# B&R Automation Studio project 305841_E00002_AM_0 (part 4)

#### Init.st
```iecst
PROGRAM _INIT

  // TODO: Security levels. For now just set as operator so OM SM can be programmed
  operatingMode.SecurityLevel := SL_OPERATOR;

  // EMO Reset time
  timeEStopResetAllow := T#10s;
  timeResetPulse := T#1s;

  // Init to create variables
  // If values are only mapped, and not used in logic anywhere, the compiler does not
  // create them. They are not available to
  // the HMI, and the compiler also complains about
  // them being declared but not used
  fs_AllSMsOk := FALSE;
  fs_EmoCmd := FALSE;
  fs_EmoOwsActive := FALSE;
  fs_EmoOwsOk := FALSE;
  // pendant signals are mapped into pendant structure
  // fs_EmoPendantActive := FALSE;
  // fs_EmoPendantOk := FALSE;
  // fs_AllowPendantMoves := FALSE;
  fs_KeyswitchInRun := FALSE;
  fs_KeyswitchOk := FALSE;
  fs_InSafeMode := FALSE;
  fs_StartPbActive := FALSE;
  fs_StartPbOk := FALSE;
  fs_StopPbActive := FALSE;
  fs_StopPbOk := FALSE;
  fs_CfGateClosedLocked := FALSE;
  fs_CfGateClosedOk := FALSE;

  ts_ResetEStop := FALSE;
  ts_ResetSafeMC := FALSE;

  // Init process req fb
  procHmiProcessReqs._I_ProcessReqs := ADR(hmiProcessReqs);
  procHmiProcessReqs._I_WpCfg := ADR(gr_CfgCurrent);
  // use the base (element 0) address for these arrays. Element
  // positions will be calculated and accessed within the function
  procHmiProcessReqs._I_pLibraryAxesReqs := ADR(hmiLibraryAxisReqs);
  procHmiProcessReqs._I_pAxis := ADR(axes);
  procHmiProcessReqs._I_pAxisPositionLimits := ADR(gr_AxisPositionLimits);

  // Init manual mode requests
  hmiLibraryAxisReqs[AD_SPINDLE].axisNo := DINT_TO_USINT(AD_SPINDLE);
  hmiMachineAxisReqs[AD_SPINDLE].axisNo := DINT_TO_USINT(AD_SPINDLE);
  hmiMachineAxisReqs[AD_SPINDLE].axisDesignation := AD_SPINDLE;
  procManualAxisReqsSpindle._I_Axis := ADR(axes[AD_SPINDLE]);
  procManualAxisReqsSpindle._I_SlaveAxis := ADR(axes[axes[AD_SPINDLE].CouplingParameters.SlaveAxisNo]);
  procManualAxisReqsSpindle._I_LibraryAxisReqs := ADR(hmiLibraryAxisReqs[AD_SPINDLE]);
  procManualAxisReqsSpindle._I_MachineAxisReqs := ADR(hmiMachineAxisReqs[AD_SPINDLE]);
  procManualAxisReqsSpindle._I_AxisPositionLimits := ADR(gr_AxisPositionLimits[AD_SPINDLE]);

  // Outer Eccentric
  hmiLibraryAxisReqs[AD_OUTER_ECCENTRIC].axisNo := DINT_TO_USINT(AD_OUTER_ECCENTRIC);
  hmiMachineAxisReqs[AD_OUTER_ECCENTRIC].axisNo := DINT_TO_USINT(AD_OUTER_ECCENTRIC);
  hmiMachineAxisReqs[AD_OUTER_ECCENTRIC].axisDesignation := AD_OUTER_ECCENTRIC;
  procManualAxisReqsOutE._I_Axis := ADR(axes[AD_OUTER_ECCENTRIC]);
  procManualAxisReqsOutE._I_SlaveAxis := ADR(axes[axes[AD_OUTER_ECCENTRIC].CouplingParameters.SlaveAxisNo]);
  procManualAxisReqsOutE._I_LibraryAxisReqs := ADR(hmiLibraryAxisReqs[AD_OUTER_ECCENTRIC]);
  procManualAxisReqsOutE._I_MachineAxisReqs:= ADR(hmiMachineAxisReqs[AD_OUTER_ECCENTRIC]);
  procManualAxisReqsOutE._I_AxisPositionLimits := ADR(gr_AxisPositionLimits[AD_OUTER_ECCENTRIC]);

  // Inner Eccentric
  hmiLibraryAxisReqs[AD_INNER_ECCENTRIC].axisNo := DINT_TO_USINT(AD_INNER_ECCENTRIC);
  hmiMachineAxisReqs[AD_INNER_ECCENTRIC].axisNo := DINT_TO_USINT(AD_INNER_ECCENTRIC);
  hmiMachineAxisReqs[AD_INNER_ECCENTRIC].axisDesignation := AD_INNER_ECCENTRIC;
  procManualAxisReqsInE._I_Axis := ADR(axes[AD_INNER_ECCENTRIC]);
  procManualAxisReqsInE._I_SlaveAxis := ADR(axes[axes[AD_INNER_ECCENTRIC].CouplingParameters.SlaveAxisNo]);
  procManualAxisReqsInE._I_LibraryAxisReqs := ADR(hmiLibraryAxisReqs[AD_INNER_ECCENTRIC]);
  procManualAxisReqsInE._I_MachineAxisReqs := ADR(hmiMachineAxisReqs[AD_INNER_ECCENTRIC]);
  procManualAxisReqsInE._I_AxisPositionLimits := ADR(gr_AxisPositionLimits[AD_INNER_ECCENTRIC]);

  // Z
  hmiLibraryAxisReqs[AD_Z].axisNo := DINT_TO_USINT(AD_Z);
  hmiMachineAxisReqs[AD_Z].axisNo := DINT_TO_USINT(AD_Z);
  hmiMachineAxisReqs[AD_Z].axisDesignation := AD_Z;
  procManualAxisReqsZ._I_Axis := ADR(axes[AD_Z]);
  procManualAxisReqsZ._I_SlaveAxis := ADR(axes[axes[AD_Z].CouplingParameters.SlaveAxisNo]);
  procManualAxisReqsZ._I_LibraryAxisReqs := ADR(hmiLibraryAxisReqs[AD_Z]);
  procManualAxisReqsZ._I_MachineAxisReqs := ADR(hmiMachineAxisReqs[AD_Z]);
  procManualAxisReqsZ._I_AxisPositionLimits := ADR(gr_AxisPositionLimits[AD_Z]);

  // Handwheel (Axis 7)
  hmiLibraryAxisReqs[AD_HANDWHEEL].axisNo := DINT_TO_USINT(AD_HANDWHEEL);
  hmiMachineAxisReqs[AD_HANDWHEEL].axisNo := DINT_TO_USINT(AD_HANDWHEEL);
  hmiMachineAxisReqs[AD_HANDWHEEL].axisDesignation := AD_HANDWHEEL;
  procManualAxisReqsHw._I_Axis := ADR(axes[AD_HANDWHEEL]);
  procManualAxisReqsHw._I_SlaveAxis := ADR(axes[axes[AD_HANDWHEEL].CouplingParameters.SlaveAxisNo]);
  procManualAxisReqsHw._I_LibraryAxisReqs := ADR(hmiLibraryAxisReqs[AD_HANDWHEEL]);
  procManualAxisReqsHw._I_MachineAxisReqs := ADR(hmiMachineAxisReqs[AD_HANDWHEEL]);
  procManualAxisReqsHw._I_AxisPositionLimits := ADR(gr_AxisPositionLimits[AD_HANDWHEEL]);

  // Cutting fluid VFD (Axis 8)
  hmiLibraryAxisReqs[AD_CF_VFD].axisNo := DINT_TO_USINT(AD_CF_VFD);
  hmiMachineAxisReqs[AD_CF_VFD].axisNo := DINT_TO_USINT(AD_CF_VFD);
  hmiMachineAxisReqs[AD_CF_VFD].axisDesignation := AD_CF_VFD;
  procManualAxisReqsCfVfd._I_Axis := ADR(axes[AD_CF_VFD]);
  procManualAxisReqsCfVfd._I_SlaveAxis := ADR(axes[axes[AD_CF_VFD].CouplingParameters.SlaveAxisNo]);
  procManualAxisReqsCfVfd._I_LibraryAxisReqs := ADR(hmiLibraryAxisReqs[AD_CF_VFD]);
  procManualAxisReqsCfVfd._I_MachineAxisReqs := ADR(hmiMachineAxisReqs[AD_CF_VFD]);
  procManualAxisReqsCfVfd._I_AxisPositionLimits := ADR(gr_AxisPositionLimits[AD_CF_VFD]);

  // Clear reqs that may result in motion or physical changes to an axis
  ClearMotionReqs;
  // Clear other requests
  ClearNonMotionReqs;

END_PROGRAM
```

#### LocalFunctions.st
```iecst
(* This function block will turn machine specific requests into GaMpMotion library requests,
and the library requests will handled with the motion library.
In this way, there is a cascading mechanism to get machine specific then axis
specific reqeusts processed by standard library functions,
even when process or machine specific things are not known by the library functions.
Note that the HMI binds to value in library axis req (sMot_HmiAxisReqs) for the move
requests, and move params. When controlling an individual axis, these are not machine specific.
This fb handles things like enable/disable choices based on selection, or other machine specific things. *)
FUNCTION_BLOCK fbHandleHmiAxisReq // Condition HMI machine specific requests, and then process them with GaMpMotion library fbProcessHmiAxisReq.
  // Map (decode) HMI move type and then direction that the GAMpMotion library will see.
  // Note the direction and move parameters allowd are be influenced by the move type.
  // Do this before processing the move request so values can be checked or used before issuing a move.

  // Endless Axes, or continuous rotary axes (spindle and eccentrics) in this case,
  // in theory can use pos, neg, or shortest path (NOT supported yet).
  // For absolute moves, but non-continuous axes (Z) don't have a specfied direction for absolute moves -- the
  // direction is inherent to the requested position.
  // Also, an absolute move does not need distance, and a relative move does not need a position.
  // A velocity move does not need either.
  // Set the enable bits of the move direction as appropriate
  IF _I_MachineAxisReqs.moveDesignation = 0 THEN // absolute
    // An absolute move does not use distance, only position
    _I_MachineAxisReqs.moveDistanceEnable := FALSE;
    _I_MachineAxisReqs.movePositionEnable := TRUE;
    // now look at the axis and decied on what directions are allowed.
    IF _I_Axis.isAxisEndless THEN
      // Endless axis, absolute move: forward, backward, and shortest (if supported) are allowed
      _I_MachineAxisReqs.directionPosEnable := TRUE;
      _I_MachineAxisReqs.directionNegEnable := TRUE;
      _I_MachineAxisReqs.directionShortestEnable := FALSE; // could be true, but shortest is not supported yet
      // If the selected direction is shortest, then clear the selection
      IF _I_MachineAxisReqs.direction = 2 THEN
        _I_MachineAxisReqs.direction := -1;
      END_IF;
    ELSE
      // For non-endless axis, direction is inferred by move position, so the operator does not choose it
      // Disable choices and clear the selection
      _I_MachineAxisReqs.directionPosEnable := FALSE;
      _I_MachineAxisReqs.directionNegEnable := FALSE;
      _I_MachineAxisReqs.directionShortestEnable := FALSE;
      _I_MachineAxisReqs.direction := -1;
    END_IF;
  ELSIF _I_MachineAxisReqs.moveDesignation = 1 THEN // relative
    // A relative move does not use position, only distance
    _I_MachineAxisReqs.moveDistanceEnable := TRUE;
    _I_MachineAxisReqs.movePositionEnable := FALSE;
    // All axes, relative move: forward and backward are viable selections
    _I_MachineAxisReqs.directionPosEnable := TRUE;
    _I_MachineAxisReqs.directionNegEnable := TRUE;
    _I_MachineAxisReqs.directionShortestEnable := FALSE;
    // If the selected direction is shortest, then clear the selection
    IF _I_MachineAxisReqs.direction = 2 THEN
      _I_MachineAxisReqs.direction := -1;
    END_IF;
  ELSIF _I_MachineAxisReqs.moveDesignation = 2 THEN // velocity
    // A velocity move does not use position or distance
    _I_MachineAxisReqs.moveDistanceEnable := FALSE;
    _I_MachineAxisReqs.movePositionEnable := FALSE;
    // All axes, velocity move: forward and backward are viable selections
    _I_MachineAxisReqs.directionPosEnable := TRUE;
    _I_MachineAxisReqs.directionNegEnable := TRUE;
    _I_MachineAxisReqs.directionShortestEnable := FALSE;
    // If the selected direction is shortest, then clear the selection
    IF _I_MachineAxisReqs.direction = 2 THEN
      _I_MachineAxisReqs.direction := -1;
    END_IF;
  ELSE
    // Not caught move type (error case).
    // Allow move direction so move type can be determined in the move velocity case
    _I_MachineAxisReqs.moveDistanceEnable := FALSE;
    _I_MachineAxisReqs.movePositionEnable := FALSE;
    _I_MachineAxisReqs.directionPosEnable := FALSE;
    _I_MachineAxisReqs.directionNegEnable := FALSE;
    _I_MachineAxisReqs.directionShortestEnable := FALSE;
    _I_MachineAxisReqs.direction := -1;
  END_IF;

  // Coordinated axis PB enable related

  // Gear In and Cam In
  // There must be a slave axis designated,
  // the axes must be homed and enabled,
  // and these two (gear/cam) are mutually exclusive of each other
  _I_MachineAxisReqs.gearInEnable :=
    _I_Axis.CouplingParameters.SlaveAxisNo <> 0 AND
    _I_Axis.Status.IsHomed AND _I_Axis.Status.IsPoweredOn AND
    _I_SlaveAxis.Status.IsHomed AND _I_SlaveAxis.Status.IsPoweredOn AND
    NOT _I_Axis.fbCamIn.Active;

  _I_MachineAxisReqs.camInEnable :=
    _I_Axis.CouplingParameters.SlaveAxisNo <> 0 AND
    _I_Axis.Status.IsHomed AND _I_Axis.Status.IsPoweredOn AND
    _I_SlaveAxis.Status.IsHomed AND _I_SlaveAxis.Status.IsPoweredOn AND
    NOT _I_Axis.fbGearIn.Active;

  // Disengage enabled if gearing or caming is active
  _I_MachineAxisReqs.disengageEnable := _I_Axis.fbGearIn.Active OR _I_Axis.fbCamIn.Active;

  // Coordinated shift commands cannot be enabled unless:
  // 1) The slave is gear coordinated and InSync
  // 2) The master is moving ?? TODO: verify
  // 3) Phase shift and offset shift are not in progress
  // 4) Cam is not active
  _I_MachineAxisReqs.shiftEnable :=
    _I_Axis.Status.IsGearInSync AND
    //_I_Axis.Status.IsMoveActive AND
    NOT _I_Axis.fbOffsetShift.ShiftStarted AND
    NOT _I_Axis.fbPhaseShift.ShiftStarted AND
    NOT _I_Axis.fbCamIn.Active;

  // Now the direction options should be qualified, set the direction that the GAMpMotion library will see
  _I_LibraryAxisReqs.Direction := fctDecodeHmiDirection(_I_DirectionReq := _I_MachineAxisReqs.direction);

  // Decode the HMI move designation into one the GAMpMotion library will see
  _I_LibraryAxisReqs.moveDesignation := fctDecodeHmiMoveType(
  _I_AxisIsEndless := _I_Axis.isAxisEndless,
  _I_MoveReq := _I_MachineAxisReqs.moveDesignation,
  _I_MoveDirection := _I_LibraryAxisReqs.Direction
  );

  // The move type and direction have now been pre-processed. Call the library function to process the requests.
  procLibraryReq(_I_HmiAxisReq := ADR(_I_LibraryAxisReqs),
                 _I_Axis := ADR(_I_Axis),
                 _I_SlaveAxis := ADR(_I_SlaveAxis),
                 _I_AxisPositionLimits := ADR(_I_AxisPositionLimits),
                 _I_ToleranceZeroDepth := TOL_DEPTH_ZERO_DEG);

END_FUNCTION_BLOCK

(* This function block will turn process requests into GaMpMotion library requests.
The GA Motion Library requests will then be handled by the library.
In this way, there is a cascading mechanism to get process specific
reqeusts processed by standard library functions, even when process specific things
are not known by the library functions.*)
FUNCTION_BLOCK fbHandleHmiProcessReqs (* Turn process specific requests into GaMpMotion library requests. *)
  // Calc structure sizes becuase they will be used several times
  szLibReq := SIZEOF(sMot_HmiAxisReqs);
  szAxis := SIZEOF(sMot_Axis);
  szAxisPosLimits := SIZEOF(sMot_PositionLimits);

  // **** Process Cutting Fluid VFD requests

  // First get the CF structures by address arithmetic
  rLibReqs ACCESS _I_pLibraryAxesReqs + (AD_CF_VFD * szLibReq);
  rAxis ACCESS _I_pAxis + (AD_CF_VFD * szAxis);

  // If the axis is enabled issue moves. Otherwise do nothing.
  // Requests get cleared at the end either way
  IF rAxis.Status.IsPoweredOn THEN
    IF _I_ProcessReqs.cfReqRun THEN
      // TODO: Incorporate pressure control
      // FOR NOW: Use RPM regardless
      IF _I_ProcessReqs.cfIsInPressureControl THEN
        rAxis.MoveParameters.Velocity := _I_ProcessReqs.cfRpmCmd / 60.0; // hmi in rpm, but axis is in rps
      ELSE
        rAxis.MoveParameters.Velocity := _I_ProcessReqs.cfRpmCmd / 60.0; // hmi in rpm, but axis is in rps
      END_IF;
      rAxis.MoveParameters.Direction := mcDIR_POSITIVE;
      rAxis.MoveParameters.Acceleration := _I_WpCfg.cfVfd.accel / 60.0; // hmi in rpm, but axis is in rps
      rAxis.MoveParameters.Deceleration := _I_WpCfg.cfVfd.decel / 60.0; // hmi in rpm, but axis is in rps
      rAxis.Commands.MoveVelocityReq := TRUE;
    END_IF;

    IF _I_ProcessReqs.cfReqStop THEN
      rAxis.MoveParameters.Deceleration := _I_WpCfg.cfVfd.decel;
      rAxis.Commands.HaltReq := TRUE;
    END_IF;

  END_IF;

  // **** Process Z axis requests
  // First get the Z structures by address arithmetic
  rLibReqs ACCESS _I_pLibraryAxesReqs + (AD_Z * szLibReq);
  rAxis ACCESS _I_pAxis + (AD_Z * szAxis);
  // get the slave number, and then calc the memory offset
  slaveNum := rAxis.CouplingParameters.SlaveAxisNo;
  rSlaveAxis ACCESS _I_pAxis + (slaveNum * szAxis);
  rAxisPositionLimits ACCESS _I_pAxisPositionLimits + (AD_Z * szAxisPosLimits);

  // Set position requests. Axis needs to be homed if current position is needed.
  // Requests get cleared at the end either way
  IF _I_ProcessReqs.zReqPosSocUseCurrent AND rAxis.Status.IsHomed THEN // home needed since axis position is used
    _I_WpCfg.zAxis.startOfCutPos := rAxis.Status.Position;
  END_IF;
  IF _I_ProcessReqs.zReqPosSocUseSpecified THEN // position specified, homing isn't needed
    _I_WpCfg.zAxis.startOfCutPos := _I_ProcessReqs.zReqPosSoc;
  END_IF;
  IF _I_ProcessReqs.zReqPosLUnLUseCurrent AND rAxis.Status.IsHomed THEN // home needed since axis position is used
    _I_WpCfg.zAxis.loadUnloadPos := rAxis.Status.Position;
  END_IF;
  IF _I_ProcessReqs.zReqPosLUnLUseSpecified THEN // position specified, homing isn't needed
    _I_WpCfg.zAxis.loadUnloadPos := _I_ProcessReqs.zReqPosLUnL;
  END_IF;

  // If the axis is enabled and homed, issue moves. Otherwise do nothing.
  // Requests get cleared at the end either way
  IF rAxis.Status.IsHomed AND rAxis.Status.IsPoweredOn THEN
    IF _I_ProcessReqs.zReqMoveUpLimit THEN
      rAxis.MoveParameters.Position := rAxisPositionLimits.PositionLimitPos;
      rAxis.MoveParameters.Velocity := _I_WpCfg.zAxis.indexSpeed;
      rAxis.MoveParameters.Acceleration := _I_WpCfg.zAxis.accel;
      rAxis.MoveParameters.Deceleration := _I_WpCfg.zAxis.decel;
      rAxis.Commands.MoveAbsoluteReq := TRUE;
    END_IF;

    IF _I_ProcessReqs.zReqMoveDownLimit THEN
      rAxis.MoveParameters.Position := rAxisPositionLimits.PositionLimitNeg;
      rAxis.MoveParameters.Velocity := _I_WpCfg.zAxis.indexSpeed;
      rAxis.MoveParameters.Acceleration := _I_WpCfg.zAxis.accel;
      rAxis.MoveParameters.Deceleration := _I_WpCfg.zAxis.decel;
      rAxis.Commands.MoveAbsoluteReq := TRUE;
    END_IF;

    IF _I_ProcessReqs.zReqMoveLUnL AND _I_WpCfg.zAxis.loadUnloadPos > 0.0 THEN
      rAxis.MoveParameters.Position := _I_WpCfg.zAxis.loadUnloadPos;
      rAxis.MoveParameters.Velocity := _I_WpCfg.zAxis.indexSpeed;
      rAxis.MoveParameters.Acceleration := _I_WpCfg.zAxis.accel;
      rAxis.MoveParameters.Deceleration := _I_WpCfg.zAxis.decel;
      rAxis.Commands.MoveAbsoluteReq := TRUE;
    END_IF;

    IF _I_ProcessReqs.zReqMoveSoc AND _I_WpCfg.zAxis.startOfCutPos > 0.0 THEN
      rAxis.MoveParameters.Position := _I_WpCfg.zAxis.startOfCutPos;
      rAxis.MoveParameters.Velocity := _I_WpCfg.zAxis.indexSpeed;
      rAxis.MoveParameters.Acceleration := _I_WpCfg.zAxis.accel;
      rAxis.MoveParameters.Deceleration := _I_WpCfg.zAxis.decel;
      rAxis.Commands.MoveAbsoluteReq := TRUE;
    END_IF;

    IF _I_ProcessReqs.zReqMoveIndexUp AND _I_WpCfg.zAxis.indexDist > 0.0 THEN
      rAxis.MoveParameters.Distance := ABS(_I_WpCfg.zAxis.indexDist); // make sure distance is positive
      rAxis.MoveParameters.Velocity := _I_WpCfg.zAxis.indexSpeed;
      rAxis.MoveParameters.Acceleration := _I_WpCfg.zAxis.accel;
      rAxis.MoveParameters.Deceleration := _I_WpCfg.zAxis.decel;
      rAxis.Commands.MoveRelativeReq := TRUE;
    END_IF;

    IF _I_ProcessReqs.zReqMoveIndexDown AND _I_WpCfg.zAxis.indexDist > 0.0 THEN
      rAxis.MoveParameters.Distance := -1.0 * ABS(_I_WpCfg.zAxis.indexDist); // make sure distance is negative
      rAxis.MoveParameters.Velocity := _I_WpCfg.zAxis.indexSpeed;
      rAxis.MoveParameters.Acceleration := _I_WpCfg.zAxis.accel;
      rAxis.MoveParameters.Deceleration := _I_WpCfg.zAxis.decel;
      rAxis.Commands.MoveRelativeReq := TRUE;
    END_IF;

  END_IF;

  // **** Process Cutting Head Requests
  // First get the Inner Eccentric structures by address arithmetic
  rLibReqs ACCESS _I_pLibraryAxesReqs + (AD_INNER_ECCENTRIC * szLibReq);
  rAxis ACCESS _I_pAxis + (AD_INNER_ECCENTRIC * szAxis);
  // get the slave number, and then calc the memory offset
  slaveNum := rAxis.CouplingParameters.SlaveAxisNo;
  rSlaveAxis ACCESS _I_pAxis + (slaveNum * szAxis);
  rAxisPositionLimits ACCESS _I_pAxisPositionLimits + (AD_INNER_ECCENTRIC * szAxisPosLimits);

  // If the axis is enabled and homed, issue moves. Otherwise do nothing.
  // Requests get cleared at the end either way
  IF rAxis.Status.IsHomed AND rAxis.Status.IsPoweredOn THEN
    IF _I_ProcessReqs.cuttingHeadMoveReqRetract THEN
      // Retract cutting head req
      IF rAxis.Status.IsGearInSync OR rAxis.Status.IsCamInSync THEN
        // Axis is coordinated. Modify the offset using the master
        ;
        // TODO: Add cases for both inner and outer stopped
        // TODO: Either or both running but not coord not supported
      END_IF;
    END_IF;
  END_IF;

  // Clear the process requests
  pSrc := ADR(_I_ProcessReqs.StartOfClearedRequests);
  pDest := ADR(_I_ProcessReqs.EndOfClearedRequests);
  byteCount := pDest - pSrc + SIZEOF(BOOL);
  nextAddr := brsmemset(pSrc, 0, byteCount);

END_FUNCTION_BLOCK

// The HMI can easily set values like 0, 1, 2 from radio buttons for example, but it is harder to set specific move type values
// This function is intended to take an HMI selection and return a move type usable by the GaMpMotion library.
// In the velocity move type case, if axis is endless, a velocity move is used. If the axis is
// not endless, jog limit instructions are used so limits can be considered.
FUNCTION fctDecodeHmiMoveType
  // Absolute move: HMI Value 0, GaMpMotion library 16#40
  // Relative move: HMI Value 1, GaMpMotion library 16#20
  // Velocity move: HMI Value 2
  // Velocity GaMpMotion library 16#10
  // Jog Limit Up Fwd GaMpMotion library 16#04
  // Jog Limit Down Rev GaMpMotion library 16#08
  IF _I_MoveReq = 0 THEN
    fctDecodeHmiMoveType := GAMOT_MD_ABSOLUTE;
  ELSIF _I_MoveReq = 1 THEN
    fctDecodeHmiMoveType := GAMOT_MD_RELATIVE;
  ELSIF _I_MoveReq = 2 THEN
    // If the axis is endless, use a velocity move, otherwise use a Jog Limit move
    // The jog limit requires a direction so the correct instruction and limit can be considered.
    IF _I_AxisIsEndless THEN
      fctDecodeHmiMoveType := GAMOT_MD_VELOCITY;
    ELSE
      IF _I_MoveDirection = mcDIR_POSITIVE THEN
        fctDecodeHmiMoveType := GAMOT_MD_JOG_LIMIT_UP_FWD;
      ELSIF _I_MoveDirection = mcDIR_NEGATIVE THEN
        fctDecodeHmiMoveType := GAMOT_MD_JOG_LIMIT_DOWN_REV;
      ELSE
        fctDecodeHmiMoveType := GAMOT_MD_NO_MOVE_COMMANDED;
      END_IF;
    END_IF;
  ELSE
      fctDecodeHmiMoveType := GAMOT_MD_NO_MOVE_COMMANDED;
  END_IF;
END_FUNCTION

// The HMI can easily set values like 0, 1, 2 from radio buttons, but it is harder to set specific move type values
// This function is intended to take an HMI selection and return a direction usable by the McAxis library
FUNCTION fctDecodeHmiDirection
  // Positive Direction: HMI Value 0, GaMpMotion library 0
  // Negative Direction: HMI Value 1, GaMpMotion library 1
  // Shortest Path:      HMI Value 2, GaMpMotion library 3
  IF _I_DirectionReq = 0 THEN
    fctDecodeHmiDirection := mcDIR_POSITIVE;
  ELSIF _I_DirectionReq = 1 THEN
    fctDecodeHmiDirection := mcDIR_NEGATIVE;
  ELSIF _I_DirectionReq = 2 THEN
    fctDecodeHmiDirection := mcDIR_SHORTEST_WAY;
  ELSE
    fctDecodeHmiDirection := mcDIR_UNDEFINED;
  END_IF;
END_FUNCTION

// The HMI can easily set values like 0, 1, 2 from radio buttons, but it is harder to set specific sub mode values.
// This function is intended to take an HMI selection and return a sub mode usable by the PLC logic.
FUNCTION fctDecodeHmiSubMode
  // Continuous:   HMI Value 0, PLC Value OM_PROD_SM_CONTINUOUS (16#40)
  // Single Cycle: HMI Value 1, PLC Value OM_PROD_SM_SINGLE (16#41)
  // Single Step:  HMI Value 2, PLC Value OM_PROD_SM_STEPPED (16#42)
  IF _I_SubModeReq = 0 THEN
    fctDecodeHmiSubMode := OM_PROD_SM_CONTINUOUS;
  ELSIF _I_SubModeReq = 1 THEN
    fctDecodeHmiSubMode := OM_PROD_SM_SINGLE;
  ELSIF _I_SubModeReq = 2 THEN
    fctDecodeHmiSubMode := OM_PROD_SM_STEPPED;
  ELSE
    fctDecodeHmiSubMode := OM_UNKNOWN;
  END_IF;
END_FUNCTION
```

#### OmSafeDev.sfc
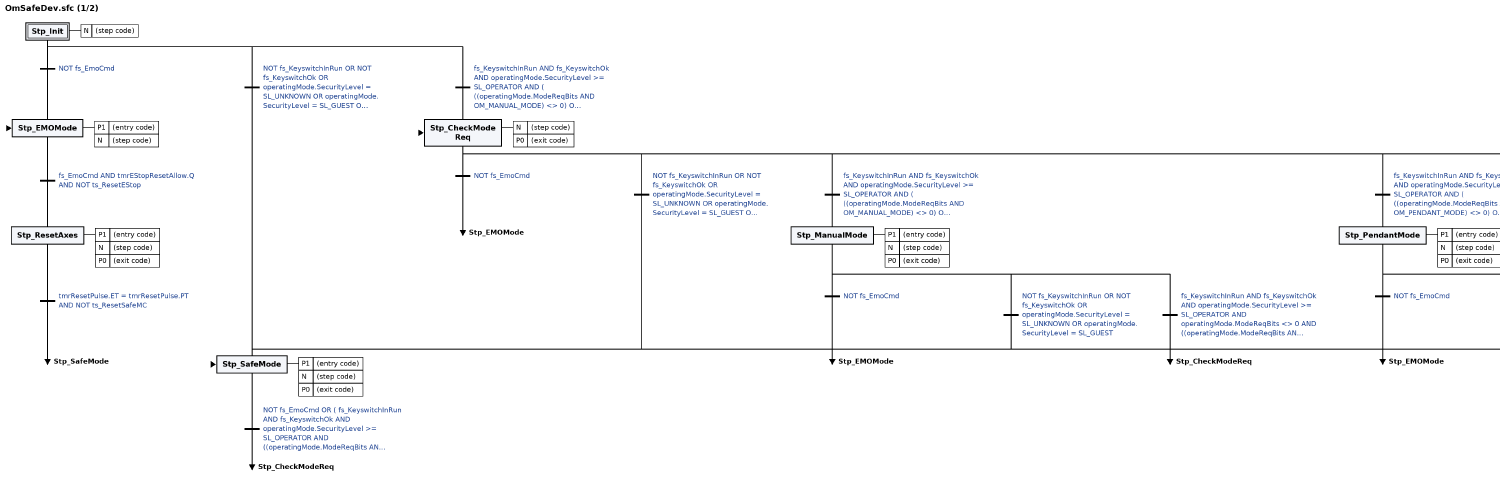
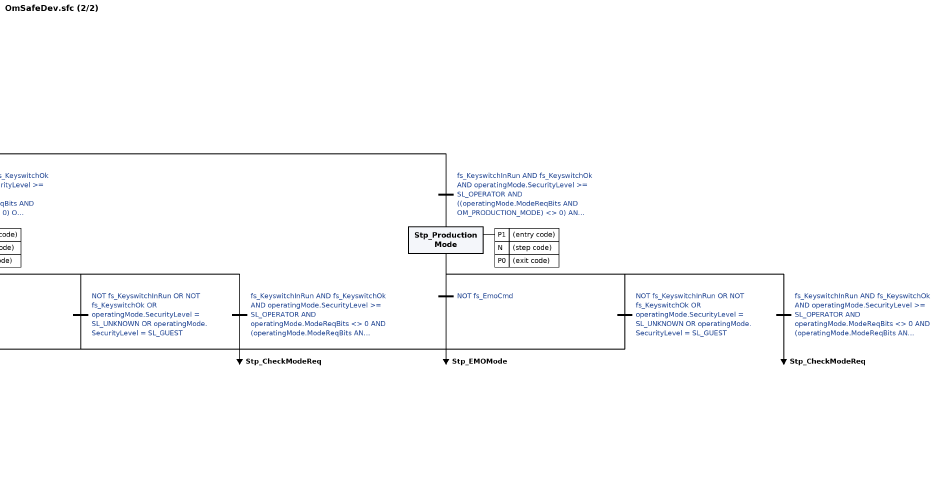
```iecst
PROGRAM _CYCLIC
INITIAL_STEP Stp_Init:
// Set Operating State
operatingMode.OperatingMode := OM_INITIAL;

END_STEP
TRANSITION EMO Cmd FROM Stp_Init TO Stp_EMOMode:=
// EStop command from safety plc H:Ok, L:EMO
NOT fs_EmoCmd
END_TRANSITION
TRANSITION keyswich in safe, not ok or bad SL or no mode req FROM Stp_Init TO Stp_SafeMode:=
// Keyswitch not in run or not okay
NOT fs_KeyswitchInRun OR
NOT fs_KeyswitchOk OR
// or not adequate security level
operatingMode.SecurityLevel = SL_UNKNOWN OR
operatingMode.SecurityLevel = SL_GUEST OR
// Or a mode isnt' being requested.
// Go to safe initially if all else is okay so a mode must be chosen
operatingMode.ModeReqBits = 0
END_TRANSITION
TRANSITION keyswitch in run and SL FROM Stp_Init TO Stp_CheckModeReq:=
// Keyswitch in run and adequate security level
fs_KeyswitchInRun AND
fs_KeyswitchOk AND
operatingMode.SecurityLevel >= SL_OPERATOR AND
// and a mode is requested
(
((operatingMode.ModeReqBits AND OM_MANUAL_MODE) <> 0) OR
((operatingMode.ModeReqBits AND OM_PENDANT_MODE) <> 0) OR
((operatingMode.ModeReqBits AND OM_PRODUCTION_MODE) <> 0)
)

END_TRANSITION
STEP Stp_CheckModeReq:
// This is a transition state. The state machine should not stay here, so don't
// set the mode upon entry. The mode in fact cannot be changed, as the current value is
// is used to transition back into the same state if a request was made but not granted
// for example production mode req but gate isn't shut.

// Clear reqs that may result in motion or physical changes to an axis
ClearMotionReqs;
// Clear other requests
ClearNonMotionReqs;

// Axis permit and other permissives
OtherModeAxisPermits;
ModeIndependentPermissions;
END_STEP
EXIT_ACTION
// Clear the request bits when leaving
operatingMode.ModeReqBits := 0;
END_ACTION
TRANSITION EMO Cmd FROM Stp_CheckModeReq TO Stp_EMOMode:=
// EStop command from safety plc H:Ok, L:EMO
NOT fs_EmoCmd
END_TRANSITION
(* @SFCISJUMP := 'Stp_EMOMode' *)
TRANSITION key not in run or bad SL or prod mode but not allowed FROM Stp_CheckModeReq TO Stp_SafeMode:=
// Keyswitch not in run or not okay, or not adequate security level
NOT fs_KeyswitchInRun OR
NOT fs_KeyswitchOk OR
operatingMode.SecurityLevel = SL_UNKNOWN OR
operatingMode.SecurityLevel = SL_GUEST OR
// or requested production mode but the gate isn't closed, so stay here in safe mode
(((operatingMode.ModeReqBits AND OM_PRODUCTION_MODE) <> 0) AND NOT fs_CfGateClosed AND operatingMode.OperatingMode = OM_SAFE_MODE)

END_TRANSITION
TRANSITION req manual mode or prod mode but not allowed FROM Stp_CheckModeReq TO Stp_ManualMode:=
// Keyswitch in run and adequate security level
fs_KeyswitchInRun AND
fs_KeyswitchOk AND
operatingMode.SecurityLevel >= SL_OPERATOR AND
(
// Req Manual Mode
((operatingMode.ModeReqBits AND OM_MANUAL_MODE) <> 0) OR
// or requested production mode but the gate isn't closed, so stay here in manual mode
(((operatingMode.ModeReqBits AND OM_PRODUCTION_MODE) <> 0) AND NOT fs_CfGateClosed AND operatingMode.OperatingMode = OM_MANUAL_MODE)
)

END_TRANSITION
STEP Stp_ManualMode:
// Block mode request for current mode, but keep the others
// This prevents it from being seen as a request
operatingMode.ModeReqBits := operatingMode.ModeReqBits AND NOT OM_MANUAL_MODE; (* bit 4 clear *)

// Axis permit and other permissives
ManualModeAxisPermits;
ModeIndependentPermissions;

// Clear process reqs
ClearProcessReqs;

// Clear production, error and estop reqs
ClearCycleReqs;

// Process manual requests
// Inputs set in init. This fb looks for a rising edge on the HMI move request, and
// one-shots the axis move requests. It is inteneded to be run on every scan,
// at least while in manual mode.
procManualAxisReqsSpindle();
procManualAxisReqsOutE();
procManualAxisReqsInE();
procManualAxisReqsZ();
procManualAxisReqsHw();
procManualAxisReqsCfVfd();
END_STEP
ENTRY_ACTION
// Set Operating State
operatingMode.OperatingMode := OM_MANUAL_MODE;
// To Safety PLC
ts_InManualMode := TRUE;

// Clear reqs that may result in motion or physical changes to an axis
ClearMotionReqs;
// Clear other requests
ClearNonMotionReqs;

// Init fb with low reqs so rising edge detection is ready
procManualAxisReqsSpindle();
procManualAxisReqsOutE();
procManualAxisReqsInE();
procManualAxisReqsZ();
procManualAxisReqsHw();
procManualAxisReqsCfVfd();
END_ACTION
EXIT_ACTION
// To Safety PLC
ts_InManualMode := FALSE;

// Clear reqs that may result in motion or physical changes to an axis
ClearMotionReqs;
// Clear other requests
ClearNonMotionReqs;

// Init fb with low reqs so rising edge detection is ready
procManualAxisReqsSpindle();
procManualAxisReqsOutE();
procManualAxisReqsInE();
procManualAxisReqsZ();
procManualAxisReqsHw();
procManualAxisReqsCfVfd();
END_ACTION
TRANSITION EMO Cmd FROM Stp_ManualMode TO Stp_EMOMode:=
// EStop command from safety plc H:Ok, L:EMO
NOT fs_EmoCmd
END_TRANSITION
(* @SFCISJUMP := 'Stp_EMOMode' *)
TRANSITION key not in run or bad SL FROM Stp_ManualMode TO Stp_SafeMode:=
// Keyswitch not in run or not okay, or not adequate security level
NOT fs_KeyswitchInRun OR
NOT fs_KeyswitchOk OR
operatingMode.SecurityLevel = SL_UNKNOWN OR
operatingMode.SecurityLevel = SL_GUEST
END_TRANSITION
TRANSITION req mode change FROM Stp_ManualMode TO Stp_CheckModeReq:=
// Keyswitch in run and adequate security level
fs_KeyswitchInRun AND
fs_KeyswitchOk AND
operatingMode.SecurityLevel >= SL_OPERATOR AND
// Req mode change (req other than current mode)
operatingMode.ModeReqBits <> 0 AND
((operatingMode.ModeReqBits AND OM_MANUAL_MODE) = 0)

END_TRANSITION
(* @SFCISJUMP := 'Stp_CheckModeReq' *)
TRANSITION req pendant mode or prod mode but not allowed FROM Stp_CheckModeReq TO Stp_PendantMode:=
// Keyswitch in run and adequate security level
fs_KeyswitchInRun AND
fs_KeyswitchOk AND
operatingMode.SecurityLevel >= SL_OPERATOR AND
(
// Req Pendant Mode
((operatingMode.ModeReqBits AND OM_PENDANT_MODE) <> 0) OR
// or requested production mode but the gate isn't closed, so stay here in pendant mode
(((operatingMode.ModeReqBits AND OM_PRODUCTION_MODE) <> 0) AND NOT fs_CfGateClosed AND operatingMode.OperatingMode = OM_PENDANT_MODE)
)

END_TRANSITION
STEP Stp_PendantMode:
// Block mode request for current mode, but keep the others
// This prevents it from being seen as a request
operatingMode.ModeReqBits := operatingMode.ModeReqBits AND NOT OM_PENDANT_MODE; (* bit 5 clear *)

// Axis permit and other permissives
PendantModeAxisPermits;
ModeIndependentPermissions;

// Clear process reqs
ClearProcessReqs;

// Clear reqs
ClearCycleReqs;

// Use the gear ratio coming from the pendant for the hmi request strucure.
// It is the hmi request structure values that will get sent to the axis.
hmiLibraryAxisReqs[AD_HANDWHEEL].gearRatioNumerator := owsPendant.GearRatioNumerator;
hmiLibraryAxisReqs[AD_HANDWHEEL].gearRatioDenominator := owsPendant.GearRatioDenominator;

// Process manual requests -- Allow these in pendant mode.
// Inputs set in init. This fb looks for a rising edge on the HMI move request, and
// one-shots the axis move requests. It is inteneded to be run on every scan,
// at least while in manual mode.
procManualAxisReqsSpindle();
procManualAxisReqsOutE();
procManualAxisReqsInE();
procManualAxisReqsZ();
procManualAxisReqsHw();
procManualAxisReqsCfVfd();

END_STEP
ENTRY_ACTION
// Set Operating State
operatingMode.OperatingMode := OM_PENDANT_MODE;
// To Safety PLC
ts_InPendantMode := TRUE;

// Disable enabled axes on entry into pendant mode -- allows starting from the same point
FOR axisNo := 1 TO AXIS_COUNT DO
  axes[axisNo].Commands.DisableReq := axes[axisNo].Status.IsPoweredOn;
END_FOR;

// Clear reqs that may result in motion or physical changes to an axis
ClearMotionReqs;
// Clear other requests
ClearNonMotionReqs;

// Init fb with low reqs so rising edge detection is ready
procManualAxisReqsSpindle();
procManualAxisReqsOutE();
procManualAxisReqsInE();
procManualAxisReqsZ();
procManualAxisReqsHw();
procManualAxisReqsCfVfd();

END_ACTION
EXIT_ACTION
// To Safety PLC
ts_InPendantMode := FALSE;

// Clear reqs that may result in motion or physical changes to an axis
ClearMotionReqs;
// Clear other requests
ClearNonMotionReqs;

// Init fb with low reqs so rising edge detection is ready
procManualAxisReqsSpindle();
procManualAxisReqsOutE();
procManualAxisReqsInE();
procManualAxisReqsZ();
procManualAxisReqsHw();
procManualAxisReqsCfVfd();
END_ACTION
TRANSITION EMO Cmd FROM Stp_PendantMode TO Stp_EMOMode:=
// EStop command from safety plc H:Ok, L:EMO
NOT fs_EmoCmd
END_TRANSITION
(* @SFCISJUMP := 'Stp_EMOMode' *)
TRANSITION key not in run or bad SL FROM Stp_PendantMode TO Stp_SafeMode:=
// Keyswitch not in run or not okay, or not adequate security level
NOT fs_KeyswitchInRun OR
NOT fs_KeyswitchOk OR
operatingMode.SecurityLevel = SL_UNKNOWN OR
operatingMode.SecurityLevel = SL_GUEST
END_TRANSITION
TRANSITION req mode change FROM Stp_PendantMode TO Stp_CheckModeReq:=
// Keyswitch in run and adequate security level
fs_KeyswitchInRun AND
fs_KeyswitchOk AND
operatingMode.SecurityLevel >= SL_OPERATOR AND
// Req mode change (req other than current mode)
operatingMode.ModeReqBits <> 0 AND
(operatingMode.ModeReqBits AND OM_PENDANT_MODE) = 0

END_TRANSITION
(* @SFCISJUMP := 'Stp_CheckModeReq' *)
TRANSITION req production mode FROM Stp_CheckModeReq TO Stp_ProductionMode:=
// Keyswitch in run and adequate security level
fs_KeyswitchInRun AND
fs_KeyswitchOk AND
operatingMode.SecurityLevel >= SL_OPERATOR AND
// Req Production Mode
((operatingMode.ModeReqBits AND OM_PRODUCTION_MODE) <> 0) AND
// gate must be closed for production mode
fs_CfGateClosed
END_TRANSITION
STEP Stp_ProductionMode:
// Block mode request for current mode, but keep the others
// This prevents it from being seen as a request
operatingMode.ModeReqBits := operatingMode.ModeReqBits AND NOT OM_PRODUCTION_MODE; (* bit 6 clear *)

// Axis permit and other permissives
ProductionModeAxisPermits;
ModeIndependentPermissions;

// Decode HMI Submode
operatingMode.SubMode := fctDecodeHmiSubMode(operatingMode.HmiSubMode);

// In production mode, cycle start/stop on PB or HMI Req, or on cycle permissives not allowed to run
// Cycle Stop
// Stop PB held in or not okay keeps req stop high - blocking the start
tmrReqStopPulse(IN:= operatingMode.HmiReqCycleStop, PT:= T#500ms);
operatingMode.ReqCycleStop := (NOT fs_StopPbOk OR NOT fs_StopPbActive OR NOT cyclePermissives.allowCycleRun) OR tmrReqStopPulse.Q; // PB is L=stop
operatingMode.HmiReqCycleStop :=FALSE;

// Cycle Start
// Stop wins if start and stop are both active.
// Start on not stop and hmi or PB press and PB Okay.
// Start PB needs to be released to get a second pulse
tmrReqStartPulse(IN:= ((operatingMode.HmiReqCycleStart OR (fs_StartPbOk AND fs_StartPbActive)) AND cyclePermissives.allowCycleRun), PT:= T#20ms);
operatingMode.ReqCycleStart := NOT operatingMode.ReqCycleStop AND tmrReqStartPulse.Q;
operatingMode.HmiReqCycleStart :=FALSE;

// Clear EMO reqs
operatingMode.ReqEmoReset := FALSE;

// process the process requests
procHmiProcessReqs();
END_STEP
ENTRY_ACTION
// Set Operating State
operatingMode.OperatingMode := OM_PRODUCTION_MODE;
// To Safety PLC
ts_InProductionMode := TRUE;
// Clear process reqs on entry -- just in case one is spuriously set
ClearProcessReqs;
END_ACTION
EXIT_ACTION
// To Safety PLC
ts_InProductionMode := FALSE;
END_ACTION
TRANSITION EMO Cmd FROM Stp_ProductionMode TO Stp_EMOMode:=
// EStop command from safety plc H:Ok, L:EMO
NOT fs_EmoCmd
END_TRANSITION
(* @SFCISJUMP := 'Stp_EMOMode' *)
TRANSITION key not in run or bad SL FROM Stp_ProductionMode TO Stp_SafeMode:=
// Keyswitch not in run or not okay, or not adequate security level
NOT fs_KeyswitchInRun OR
NOT fs_KeyswitchOk OR
operatingMode.SecurityLevel = SL_UNKNOWN OR
operatingMode.SecurityLevel = SL_GUEST
END_TRANSITION
TRANSITION req mode change FROM Stp_ProductionMode TO Stp_CheckModeReq:=
// Keyswitch in run and adequate security level
fs_KeyswitchInRun AND
fs_KeyswitchOk AND
operatingMode.SecurityLevel >= SL_OPERATOR AND
// Req mode change (req other than current mode)
operatingMode.ModeReqBits <> 0 AND
(operatingMode.ModeReqBits AND OM_PRODUCTION_MODE) = 0

END_TRANSITION
(* @SFCISJUMP := 'Stp_CheckModeReq' *)
STEP Stp_SafeMode:
// Clear mode requests if not ready to leave -- this guards against a lingering req
// being acted on long after it was issued, once conditions become okay to leave
IF NOT fs_KeyswitchInRun OR
    NOT fs_KeyswitchOk OR
    operatingMode.SecurityLevel < SL_OPERATOR THEN // OR
    // NOT fs_CfGateClosed THEN
  operatingMode.ModeReqBits := 16#0;
END_IF;

// Clear reqs that may result in motion or physical changes to an axis
ClearMotionReqs;
// Allow the other reqs (resets and set limits)

// Axis permit and other permissives
OtherModeAxisPermits;
ModeIndependentPermissions;

// Clear the other HMI Reqs
ClearCycleReqs;

END_STEP
ENTRY_ACTION
// Set Operating State
operatingMode.OperatingMode := OM_SAFE_MODE;
// To Safety PLC
ts_InSafeMode := TRUE;
// Initially clear the mode requests.
// They will be allowed once in the mode, and the keyswitch is in the run position
operatingMode.ModeReqBits := 16#0;

END_ACTION
EXIT_ACTION
// To Safety PLC
ts_InSafeMode := FALSE;
END_ACTION
TRANSITION EMO or Run and Mode Req FROM Stp_SafeMode TO Stp_CheckModeReq:=
// EStop command from safety plc H:Ok, L:EMO
NOT fs_EmoCmd OR
(
// Keyswitch in run and adequate security level
fs_KeyswitchInRun AND
fs_KeyswitchOk AND
operatingMode.SecurityLevel >= SL_OPERATOR AND
// Req Another Mode
// Leaving out of safe or emo will lock the gate,
// but the latched check is for production mode only.
((operatingMode.ModeReqBits AND OM_MANUAL_MODE) <> 0) OR
((operatingMode.ModeReqBits AND OM_PENDANT_MODE) <> 0) OR
((operatingMode.ModeReqBits AND OM_PRODUCTION_MODE) <> 0)
)

END_TRANSITION
(* @SFCISJUMP := 'Stp_CheckModeReq' *)
STEP Stp_EMOMode:

// clear mode requests while in EMO
operatingMode.ModeReqBits := 16#0;

// Axis permit and other permissives
OtherModeAxisPermits;
ModeIndependentPermissions;

// Clear reqs that may result in motion or physical changes to an axis
ClearMotionReqs;
// Clear other requests
ClearNonMotionReqs;

// Block cycle start/stop req in Emo
operatingMode.ReqCycleStart := FALSE;
operatingMode.ReqCycleStop := FALSE;
// Clear the reqs, but allow the EMO/Axis Reset ... they get handled below
operatingMode.HmiReqCycleStart := FALSE;
operatingMode.HmiReqCycleStop := FALSE;

// Run emo allow timer
// Only allow resets to emo if this timer is expired.
// If an e-stop removes power from the drives, it is bad for the drive power supplies to be
// energized less than 2 minutes after being deenergized -- capacitor discharge/recharge issue
tmrEStopResetAllow(IN:= TRUE);

// Clear the EMO reset bit if within this time
IF NOT tmrEStopResetAllow.Q THEN
  operatingMode.ReqEmoReset := FALSE;
END_IF;

// Calc how many seconds remain before a reset is allowed
eStopResetAllowSecRemain := TIME_TO_DINT(timeEStopResetAllow - tmrEStopResetAllow.ET) / 1000;

// We can't leave this state until EMO is clear, but we need the reset pulse to clear the EMO.
// If a reset request is received, send a reset pulse to the safe controller. In the event of
// multiple emo events, this may or may not clear all of them, but the status on the HMI should
// be updated, allowing the operators to see what else is needed.
// Run the reset pulse and send the reset req
tmrResetPulse(IN:= operatingMode.ReqEmoReset, PT:= timeResetPulse);
ts_ResetEStop := tmrResetPulse.Q;
operatingMode.ReqEmoReset := FALSE;

END_STEP
ENTRY_ACTION
// Set Operating State
operatingMode.OperatingMode := OM_EMO_MODE;

// To safety PLC
ts_InEmoMode := TRUE;

// Reset emo allow timer
tmrEStopResetAllow(IN:= FALSE, PT := timeEStopResetAllow);

END_ACTION
TRANSITION no emo, allow time done and reset req FROM Stp_EMOMode TO Stp_ResetAxes:=
// No more EMO, reset allow timer has expired, reset pulse is done
fs_EmoCmd AND
tmrEStopResetAllow.Q AND
// Use the reset pulse to the safe controller being done as time to leave instead of the request.
// This allows a request to create a pulse, and then be cleared.
// Meanwhile, the EMO may or may not clear, and the reset pulse will go away. If the EMO is gone
// when the reset pulse goes away, we can leave.
NOT ts_ResetEStop
END_TRANSITION
STEP Stp_ResetAxes:
// Clear mode requests while in EMO
operatingMode.ModeReqBits := 16#0;

// Run the reset pulse and send the reset req
tmrResetPulse(IN:= TRUE, PT:= timeResetPulse);
ts_ResetSafeMC := tmrResetPulse.Q;

END_STEP
ENTRY_ACTION
// Reset pulse timer
tmrResetPulse(IN:= FALSE, PT:= timeResetPulse);
END_ACTION
EXIT_ACTION
// To safety PLC
ts_InEmoMode := FALSE;

// Clear reqs that may result in motion or physical changes to an axis
ClearMotionReqs;
// Clear other requests
ClearNonMotionReqs;

// Clear other reqs
ClearCycleReqs;

END_ACTION
TRANSITION axis reset pulse done FROM Stp_ResetAxes TO Stp_SafeMode:=
// Emo Reset pulse complete
tmrResetPulse.ET = tmrResetPulse.PT AND NOT ts_ResetSafeMC
END_TRANSITION
(* @SFCISJUMP := 'Stp_SafeMode' *)
END_PROGRAM
```

### Program Logical/PlcLogic/Annunc (IEC)

#### Annunc.var - Local variables
```iecst
VAR
	tmr025Hz : TON; (* 0.25 Hz timer *)
	tmr050Hz : TON; (* 0.50 Hz timer *)
	tmr100Hz : TON; (* 1 Hz timer *)
END_VAR
```

#### Main.st - Init, cyclic, exit code
```iecst
PROGRAM _INIT
  tmr025Hz.PT := T#250ms;
  tmr050Hz.PT := T#500ms;
  tmr100Hz.PT := T#1000ms;
END_PROGRAM

PROGRAM _CYCLIC

  // Create blinking bits (global variables), 50% duty cycle
  // 0.25 Hz (4x/sec)
  tmr025Hz(IN:= NOT tmr025Hz.Q);
  IF tmr025Hz.Q THEN
    blink025Hz := NOT blink025Hz;
  END_IF;
  // 0.5 Hz (2x/sec)
  tmr050Hz(IN:= NOT tmr050Hz.Q);
  IF tmr050Hz.Q THEN
    blink050Hz := NOT blink050Hz;
  END_IF;
  // 1.0 Hz (1x/sec)
  tmr100Hz(IN:= NOT tmr100Hz.Q);
  IF tmr100Hz.Q THEN
    blink100Hz := NOT blink100Hz;
  END_IF;

  // Light the 480 VAC Okay lamp on the OWS if the power monitor in the MCP is okay.
  DO_PL_OWSAmber :=  DI_JI_480VACOk.Value;

  // **** Green Ready lamp, Green Start lamp, Red Stop lamp ****
  // Green ready lamp
  //    ON: Production mode and permissives met to run OR production mode, allowed to run and in cycle
  // Green Start Lamp
  //    ON: In production mode, start permissives met, and not in cycle. Lit indicating a press will start cycle
  //    BLINK: in production mode, and in cycle, and in cycle hold. Lit blinking indicating a press will continue cycle
  // Red Stop lamp
  //    ON: In production mode and in cycle. Lit indicating a press will stop cycle.
  //    BLINK: In production mode and cycle is stopping.
  DO_PL_OWSGreen :=
      (operatingMode.OperatingMode = OM_PRODUCTION_MODE AND cyclePermissives.allowCycleStart) OR
      (operatingMode.OperatingMode = OM_PRODUCTION_MODE AND cyclePermissives.allowCycleRun AND operatingMode.isInCycle);

  DO_PB_OWSGreen :=
      (operatingMode.OperatingMode = OM_PRODUCTION_MODE AND cyclePermissives.allowCycleStart AND NOT operatingMode.isInCycle) OR
      (operatingMode.OperatingMode = OM_PRODUCTION_MODE AND cyclePermissives.allowCycleRun AND operatingMode.isInCycle AND operatingMode.isInCycleHold AND blink100Hz);

  DO_PB_OWSRed :=
      (operatingMode.OperatingMode = OM_PRODUCTION_MODE AND operatingMode.isInCycle AND NOT operatingMode.isStopping) OR
      (operatingMode.OperatingMode = OM_PRODUCTION_MODE AND operatingMode.isInCycle AND operatingMode.isStopping AND blink100Hz);

END_PROGRAM

PROGRAM _EXIT
	(* Insert code here *)

END_PROGRAM
```

### Program Logical/PlcLogic/AxEnable (IEC)

#### AxEnable.st
```iecst
PROGRAM _INIT

END_PROGRAM

PROGRAM _CYCLIC

  // TODO: Decide when drives shall be enabled by the PLC
  // For now, enable them for easy initial testing.
  // H: Enable, L: Stop
  axes[AD_SPINDLE].Commands.PlcSafetyEnable := TRUE;
  axes[AD_OUTER_ECCENTRIC].Commands.PlcSafetyEnable := TRUE;
  axes[AD_INNER_ECCENTRIC].Commands.PlcSafetyEnable := TRUE;
  axes[AD_Z].Commands.PlcSafetyEnable := TRUE;
  axes[AD_CF_VFD].Commands.PlcSafetyEnable := TRUE;

END_PROGRAM

PROGRAM _EXIT
	(* Insert code here *)

END_PROGRAM
```

### Program Logical/PlcLogic/ProdCycle (IEC)

#### ProdCycle.typ
```iecst
TYPE
  ePROD_CYCLE_STEP :
    (
    PCS_UNKNOWN         := 0,
    PCS_INIT            := 1,
    PCS_MODE_CHECK      := 2,
    PCS_WAIT_FOR_PROD   := 3,
    PCS_WAIT_FOR_START  := 4,
    PCS_DECOUPLE_ECC    := 5,
    PCS_RESET_AXES      := 6,
    PCS_ENABLE_AXES     := 7,
    PCS_ZERO_DEPTH      := 8,
    PCS_Z_TO_SOC        := 9,
    PCS_NEXT_CYCLE      := 10,
    PCS_START_SPINDLE   := 11,
    PCS_COUPLE_ECC      := 12,
    PCS_START_PASS      := 13,
    PCS_SYNCHING1       := 14,
    PCS_SYNCHING2       := 15,
    PCS_SYNCHING3       := 16,
    PCS_AXES_SYNCHED    := 17,
    PCS_SET_NEXT_PASS   := 18,
    PCS_SET_FINISH_PASS := 19,
    PCS_SET_RETRACT     := 20,
    PCS_STOP_SPINDLE    := 21,
    PCS_INDEX_Z_WAIT    := 22,
    PCS_CF_OFF1         := 23,
    PCS_CF_OFF2         := 24,
    PCS_Z_TO_UNLOAD     := 25,
    PCS_DONE_WAIT       := 26,
    PCS_INDEX_Z         := 27,
    PCS_EOC_WAIT        := 28,
    PCS_CF_TO           := 29,
    PCS_START_CF2       := 30,
    PCS_CYCLE_STOP      := 31,
    PCS_CS_STOP_AXES    := 32,
    PCS_CS_ZERO_DEPTH   := 33,
    PCS_CS_STOP_SPINDLE := 34,
    PCS_CS_DISABLE_AXES := 35,
    PCS_CS_STOP_CF      := 36
  ) := PCS_INIT;

  (* motion params derrived from machine/part config and process point *)
  sPartMotion : STRUCT
    warnAdjAngleTooSmall : BOOL; (* H: depth adj angle too small for fee rate and/or cutting depth *)
    totalIndexes : USINT; (* number of Z Indexes needed to process a part *)
    prodCycleStepCurrent : ePROD_CYCLE_STEP; (* last completed production cycle step *)
    passDepth : REAL; (* mm. cut pass depth *)
    cutVelocity : REAL; (* deg/sec. Inner and Outer Eccentric velocity while cutting *)
    depthAdjVelocity : REAL; (* deg/sec. **Average/Approx** velocity when adjusting depth. For infomation purposes only. *)
    depthAdjAngle : LREAL; (* degrees. Adjusted angle over which to adjust the cutting depth (i.e. offset angle). LREAL to be compatible with motion positions *)
    depthAdjAngleMin : LREAL; (* degrees. Calculated minimum adj angle given a feed rate, offset angle -- can't overspeed the inner axis (constrained by inner axis max vel *)
    passOffsetAngle : LREAL; (* +/-180 deg, +: I leads O, -: O leads I. LREAL to be compatible with motion positions *)
    finishPassOffsetAngle :  LREAL; (* +/-180 deg, +: I leads O, -: O leads I. LREAL to be compatible with motion positions  *)
    passDistance : LREAL; (* degrees. pass move distance, including starting depth adjust, and overcut. LREAL to be compatible with motion positions *)
    startOfPassPosition : LREAL; (* Where did this pass start. LREAL to be compatible with motion positions *)
    endOfPassPosition : LREAL; (* degrees calculated position at end of the pass. LREAL to be compatible with motion positions *)
    calcNextAdjPosition : LREAL; (* azimuth point where the next adjusment completes. LREAL to be compatible with motion positions *)
    calcNextAdjDistance : LREAL; (* degrees. Need to travel this far before setting up the next adjustment. LREAL to be compatible with motion positions *)
    passDistanceTraveled : LREAL; (* degrees. How far have we traveled during this pass. LREAL to be compatible with motion positions *)
  END_STRUCT;

 END_TYPE
```

#### ProdCycle.var
```iecst
VAR CONSTANT

END_VAR

VAR RETAIN
  partMotion : sPartMotion; (* calculated values for processing part. Retain to preserve dynamic values *)

END_VAR

VAR
  disableStepTO : BOOL := FALSE;
  startCycleOS : BOOL := FALSE;
  idx : SINT;

  calcReal1 : REAL;  (* temporary value *)
  calcLReal1 : LREAL; (* temporary value *)
  calcDint1 : DINT;  (* temporary value *)
  tmrStepMin : TON; (* hold step for min time *)
  tmrStepTO : TON; (* step timeout timer *)
  tmrCfShutoff : TON; (* shutoff cooling pump after a delay *)
  fbCalcMoveTimes : fbCalcTrapMoveTime; (* function block to calculate trapazoidal move times *)

  (* info to safety controller *)
  ts_InCycle : BOOL; (* tell the safe controller we are in cycle *)
  ts_cfLockGate : BOOL; (* lock the cutting fluid gate *)

  (* production cycle step information *)
  (* indexes correspond to ePROD_CYCLE_STEP values *)
  stepETs  : ARRAY[0..40] OF TIME; (* step elapsed times *)
  stepTOs  : ARRAY[0..40] OF TIME; (* step Timeout values *)
  stepIsTO : ARRAY[0..40] OF BOOL; (* set if the step has a TO *)

  prodCycleStep : ePROD_CYCLE_STEP;
END_VAR
```

#### Actions.st
```iecst
ACTION CalcPartMotion :

  // Calc cut velocity
  CalcCutVelocity;

  // Calc pass depth
  CalcPassDepth;
  // Calc the axis offset angles, in degrees, for a nominal pass and a finishing pass.
  // First calc the depth of a nominal pass, taking into account the finishing pass depth.
  // Then calc the offset angles needed to acheive the depths.
  // Note: this will enforce a minimum adjustement angle -- can't overspeed inner eccentric for a
  // given feed rate (cut velocity), cutting depth, and ajustment angle.
  // The velocity margin can be approximate by comparing partMotion.depthAdjVelocity with the
  // inner axis max velocity, axes[AD_INNER_ECCENTRIC].MoveParameters.VelocityMax.
  // Note: Before calculating the angles, this needs cut velocity to be calculated from feed rate,
  // and pass depth to be calculated from total depth and pass count.
  CalcAngles;

  // Calc depth adjustment velocity.
  // Note this is an average/approximate value for informaitional and approximate use.
  // It does not take into account accel and decel and isn't the exact value the system calculates
  // for coordinated moves.
  CalcDepthAdjVelocity;

  // Calc the number of indexes needed to process a part
  CalcTotalZIndexes;

  // Calc index related values
  CalcZIndex;

END_ACTION

ACTION CalcCutVelocity : // Calc cut velocity in deg/sec from the inside diameter and feed rate
  partMotion.cutVelocity := fctCalcCutVelocity(
  _I_InnerDiameter := gr_PartCurrent.partDfn.nomId,
  _I_FeedRate := gr_CfgCurrent.cuttingHead.feedRate);
END_ACTION

ACTION CalcPassDepth: // Calc pass depth from total depth, number of passes, and finishing pass depth
// Factor in finishing pass
  IF gr_CfgCurrent.cuttingHead.finishingPass THEN
    calcReal1 := MAX(gr_CfgCurrent.cuttingHead.finishingPassDepth, 0.0); // no negative depths
  ELSE
    calcReal1 := 0.0;
  END_IF;

  partMotion.passDepth := fctCalcPassDepth(
  _I_TotalDepth := gr_CfgCurrent.cuttingHead.totalDepth,
  _I_PassCount := gr_CfgCurrent.cuttingHead.passCount,
  _I_FPDepth := calcReal1 ); // calcReal1 at call time has the finishing pass depth
END_ACTION

ACTION CalcAngles :
  // Calc the axis offset angle in degrees given the desired cutting depth
  // Calc the angle from the calculated pass depth
  partMotion.passOffsetAngle := fctCalcAngleFromDepth(
  _I_Depth := partMotion.passDepth);

  // Calc the angle from the configured finish pass depth
  partMotion.finishPassOffsetAngle := fctCalcAngleFromDepth(
  _I_Depth := gr_CfgCurrent.cuttingHead.finishingPassDepth);

  // For a combination of offset angle, max inner axis velocity, and cut velocity, there is a minimum adjustment angle that needs to be adhered to.
  // Inner Axis Velocity = (offset angle / adj angle) * cut velocity. The cut velocity and offset angle are essentially fixed by the process settings,
  // and the inner axis velocity has an upper limit. So this means that for a given cut velocity or feed rate, there is a minimum adjustment angle.
  // Solving the eqn for adj angle ==> Adj Angle Min = (Offset Angle / Max Inner Velocity * Cut Velocity
  // Give a small margin to help prevent problems
  partMotion.depthAdjAngleMin := 1.1 * ((ABS(partMotion.passOffsetAngle) / axes[AD_INNER_ECCENTRIC].MoveParameters.VelocityMax) * partMotion.cutVelocity);
  // If the entered depth adjustment angle is too small, set the warning and enforce the minimum
  partMotion.warnAdjAngleTooSmall := gr_CfgCurrent.cuttingHead.depthAdjAngle < partMotion.depthAdjAngleMin;
  partMotion.depthAdjAngle := MAX(gr_CfgCurrent.cuttingHead.depthAdjAngle, partMotion.depthAdjAngleMin);

  // INITIALLY HARD CODE depth adj angle
  partMotion.depthAdjAngle := 10.0;

END_ACTION

ACTION CalcDepthAdjVelocity : // deg/sec. Calc depth adjustment velocity
  // Velocity of the relative eccentric motion to acheive the offset angle during the depth adj angle
  partMotion.depthAdjVelocity := fctCalcDepthAdjVelocity(
  _I_CutVelocity:= partMotion.cutVelocity,
  _I_DepthAdjAngle:= partMotion.depthAdjAngle,
  _I_OffsetAngle := partMotion.passOffsetAngle);
END_ACTION

ACTION CalcTotalZIndexes :
  // Number of indexes to process a part
  // Round up if a partial index is needed
  IF gr_PartCurrent.partDfn.nomCutLength > 0.0 AND gr_CfgCurrent.zAxis.indexDist > 0.0 THEN
    partMotion.totalIndexes := LREAL_TO_USINT(fctLRCeiling(gr_PartCurrent.partDfn.nomCutLength / gr_CfgCurrent.zAxis.indexDist));
  ELSE
    partMotion.totalIndexes := 0;
  END_IF;
END_ACTION

ACTION CalcZIndex :
  // If Z is calibrated, then see where we are for a Z index based on position.
  // Set part current isZIndexed if Z is in an index position.
  // The stat of cut position is subtracted out, and when the head is at
  // the start of cut position, the index should be 1.
  // The general algorithm is index = ((pos - start of cut) / index distance) + 1
  // An
  IF gr_PartCurrent.isZCalibrated THEN
    // Need to know position relative to the start of cut position
    calcLReal1 := axes[AD_Z].Status.Position - gr_CfgCurrent.zAxis.startOfCutPos;
    // Get the Z index count. Value of 0 means the Z position is below the start of cut position, or
    // above the cut length of the workpiece (start of cut pos + cut length, e.g. load/unload position)
    // This is a floating point number that should have a very close to an integer when Z is properly indexed
    IF calcLReal1 < (-1.0 * TOL_ZINDEX) THEN
      // If we are more negative than the tolerance, we are below the start
      // Make the index 0, and call it not indexed
      gr_PartCurrent.zIndexLRCount := 0.0;
      gr_PartCurrent.zIndexCount := 0;
      gr_PartCurrent.isZIndexed := FALSE;
    ELSIF calcLReal1 > (gr_CfgCurrent.zAxis.startOfCutPos + (gr_CfgCurrent.zAxis.indexDist * (partMotion.totalIndexes - 1))) THEN
      // If we are higher than the last index position , we are off the top end.
      // Subtract 1 from totalIndexed, because the Start of Cut is index 1, and there are total indexes - 1 above that.
      // Make the index 0, and call it not indexed
      gr_PartCurrent.zIndexLRCount := 0.0;
      gr_PartCurrent.zIndexCount := 0;
      gr_PartCurrent.isZIndexed := FALSE;
    ELSE
      // If we get here, we are somewhere within the cut length. Consider it indexed if we are at an indexed position.
      gr_PartCurrent.zIndexLRCount := (calcLReal1 / gr_CfgCurrent.zAxis.indexDist) + 1.0;  // Float value for info. SOC is 1, not zero, so we need to add 1
      gr_PartCurrent.zIndexCount := LREAL_TO_USINT(gr_PartCurrent.zIndexLRCount); // Integer index pos, rounded
      // If the position is close enough to an integer index pos, consider us indexed.
      // (Pos - SOC) - the indexed pos from SOC has to be < tolerance
      // TODO: Figure out proper index tolerance. Should correspond to needed Z index precision.
      gr_PartCurrent.isZIndexed := ABS(calcLReal1 - ((gr_PartCurrent.zIndexCount - 1) * gr_CfgCurrent.zAxis.indexDist)) < TOL_ZINDEX;
    END_IF;
  ELSE
    // Not calibrated, so no valid count and not indexed
    gr_PartCurrent.zIndexLRCount := 0.0;
    gr_PartCurrent.zIndexCount := 0;
    gr_PartCurrent.isZIndexed := FALSE;
  END_IF;

END_ACTION
```
